// TIA Portal V18 export
DATA_BLOCK "SS1_CPU1214_DI_Vars"   // DB11013
{ S7_Optimized_Access := 'FALSE' }
VERSION : 0.1
// stored: AutoNumber false, DBAccessibleFromOPCUA true, IsOnlyStoredInLoadMemory false, IsWriteProtectedInAS false
   VAR
      DI1 : "UDT_DIadv";   // HS Режим роботи "Зима"
      DI2 : "UDT_DIadv";   // HS Режим роботи "Авто"
      DI3 : "UDT_DIadv";   // HS Відмова Котел 1
      DI4 : "UDT_DIadv";   // HS Відмова Котел 2
      DI5 : "UDT_DIadv";   // HS Норм. рівень води Котел 1 (10.80)
      DI6 : "UDT_DIadv";   // HS Низький тиск Котел 1 (10.71)
      DI7 { S7_SetPoint := 'True'} : "UDT_DIadv";   // HS Високий тиск Котел 1 (10.72)
      DI8 { S7_SetPoint := 'True'} : "UDT_DIadv";   // HS Норм. рівень води Котел 2 (10.81)
      DI9 { S7_SetPoint := 'True'} : "UDT_DIadv";   // HS Низький тиск Котел 1 (10.73)
      DI10 { S7_SetPoint := 'True'} : "UDT_DIadv";   // HS Високий тиск Котел 1 (10.74)
      DI11 { S7_SetPoint := 'True'} : "UDT_DIadv";   // Резерв
      DI12 { S7_SetPoint := 'True'} : "UDT_DIadv";   // Резерв
      DI13 { S7_SetPoint := 'True'} : "UDT_DIadv";   // Резерв
      DI14 { S7_SetPoint := 'True'} : "UDT_DIadv";   // Резерв
   END_VAR
BEGIN
   DI1.cFuncSystemID := 3;
   DI1.cFuncVar := 19;
   DI2.cFuncSystemID := 3;
   DI2.cFuncVar := 8;
   DI3.cFuncSystemID := 3;
   DI3.cFuncVar := 9;
   DI4.cFuncSystemID := 3;
   DI4.cFuncVar := 20;
   DI5.cFuncSystemID := 3;
   DI5.cFuncVar := 7;
   DI6.cFuncSystemID := 3;
   DI6.cFuncVar := 21;
   DI8.cFuncSystemID := 10;
   DI8.cFuncVar := 41;
   DI9.cFuncSystemID := 10;
   DI9.cFuncVar := 43;
   DI10.cFuncSystemID := 3;
   DI10.cFuncVar := 16;
   DI11.cFuncSystemID := 0;
   DI11.cFuncVar := 0;
   DI12.cFuncSystemID := 0;
   DI12.cFuncVar := 0;
   DI13.cFuncSystemID := 0;
   DI13.cFuncVar := 0;
END_DATA_BLOCK
